FUNCTION_BLOCK FB_Roboter
VAR_INPUT
END_VAR
VAR_OUTPUT
END_VAR
VAR
END_VAR

END_FUNCTION_BLOCK

(* stored: Version 1.1.0.1, ProductVersion 3.1.4024.15
   POU FB_Roboter: Id {98968849-8f50-4fb2-866e-dc1c8bbe7081}, SpecialFunc None *)
